# EPICS autosave request: iocBoot/ioc13bmc_DAC_XPS/auto_positions.req
file "CARS_motor_positions.req",         P=$(P), M=m71
file "CARS_motor_positions.req",         P=$(P), M=m72
file "CARS_motor_positions.req",         P=$(P), M=m73
file "CARS_motor_positions.req",         P=$(P), M=m74
file "CARS_motor_positions.req",         P=$(P), M=m75
